(* Logix 5000 project; controller Just_Keyence_Vision vendor 1 type 14 code 155 rev 20.12; software revision 20.01 *)

TASK MainTask (continuous, watchdog 500 ms) : MainProgram

MODULES
   Local : vendor 1 type 14 code 155 (PointIO 0, rev 20.12)
      XG_7702 : ETHERNET-MODULE (Ethernet 192.168.1.6, rev 1.1, Output RPI 10 ms)
       : 1734-IE2V (PointIO 2, rev 3.1, Input RPI 80 ms)
      Discrete_IO : Embedded (PointIO 1, rev 20.11, Output RPI 20 ms)
       : 1734-OE2V (PointIO 3, rev 3.1, Output RPI 80 ms)
END_MODULES

PROGRAM MainProgram   (* main routine MainRoutine *)
VAR
   Timer1 : TIMER := (PRE := 1000);
   Timer2 : TIMER := (PRE := 1000);
END_VAR

ROUTINE MainRoutine   (* ladder *)
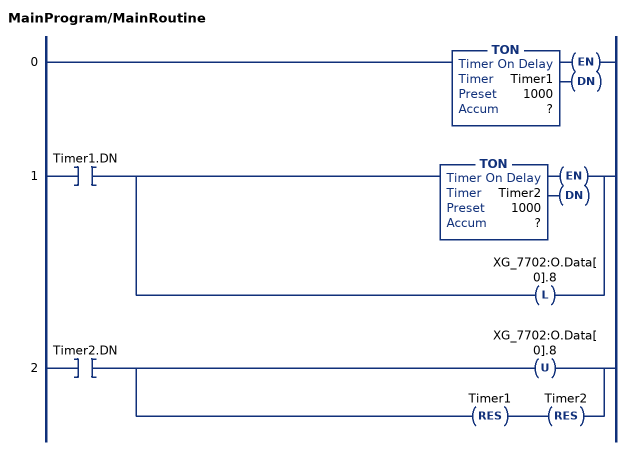
   0: TON(Timer1,?,?);
   1: XIC(Timer1.DN)[TON(Timer2,?,?) ,OTL(XG_7702:O.Data[0].8) ];
   2: XIC(Timer2.DN)[OTU(XG_7702:O.Data[0].8) ,RES(Timer1) RES(Timer2) ];
END_ROUTINE
END_PROGRAM
